// TIA Portal V17 export
// export: Created 2023-08-26T15:31:22.9849218Z, ExportSetting WithDefaults, DisplayName Totally Integrated Automation Portal, DisplayVersion V17 Update 5, DisplayName TIA Portal Openness, DisplayVersion V17 Update 5, DisplayName TIA Portal Teamcenter Gateway, DisplayVersion V17 Update 5, DisplayName TIA Portal Version Control Interface, DisplayVersion V17, DisplayName Simotion SCOUT TIA, DisplayVersion 5.4.3.0, DisplayName TIA Portal Test Suite Advanced, DisplayVersion V17 Update 1, DisplayName SIMOCODE ES, DisplayVersion V17 Update 5, DisplayName SINAMICS Startdrive Advanced, DisplayVersion V17 SP1, DisplayName SINAMICS Startdrive G130, G150, S120, S150, SINAMICS MV, S210, DisplayVersion V17 SP1, DisplayName SINAMICS Startdrive G110M, G120, G120C, G120D, G120P, G115D, DisplayVersion V17 SP1, DisplayName SIRIUS Safety ES, DisplayVersion V17 Update 5, DisplayName STEP 7 Professional, DisplayVersion V17 Update 5, DisplayName STEP 7 CFC, DisplayVersion V17 Update 1, DisplayName STEP 7 Safety, DisplayVersion V17, DisplayName WinCC Advanced, DisplayVersion V17 Update 5, DisplayName SIMATIC Visualization Architect, DisplayVersion V17 Update 5
FUNCTION "00_Only for Commissioning" : Void   // FC1, F_LAD
{ S7_Optimized_Access := 'TRUE' }
VERSION : 0.1
// Management of bypass to use during commissioning
// stored: AutoNumber true, IsIECCheckEnabled false, UDAEnableTagReadback false
BEGIN

REGION Network 1: FIRE ALARM BYPASS
   // One network per node
   // TRUE if the node is not ready to be used
   // FALSE if the node is ready
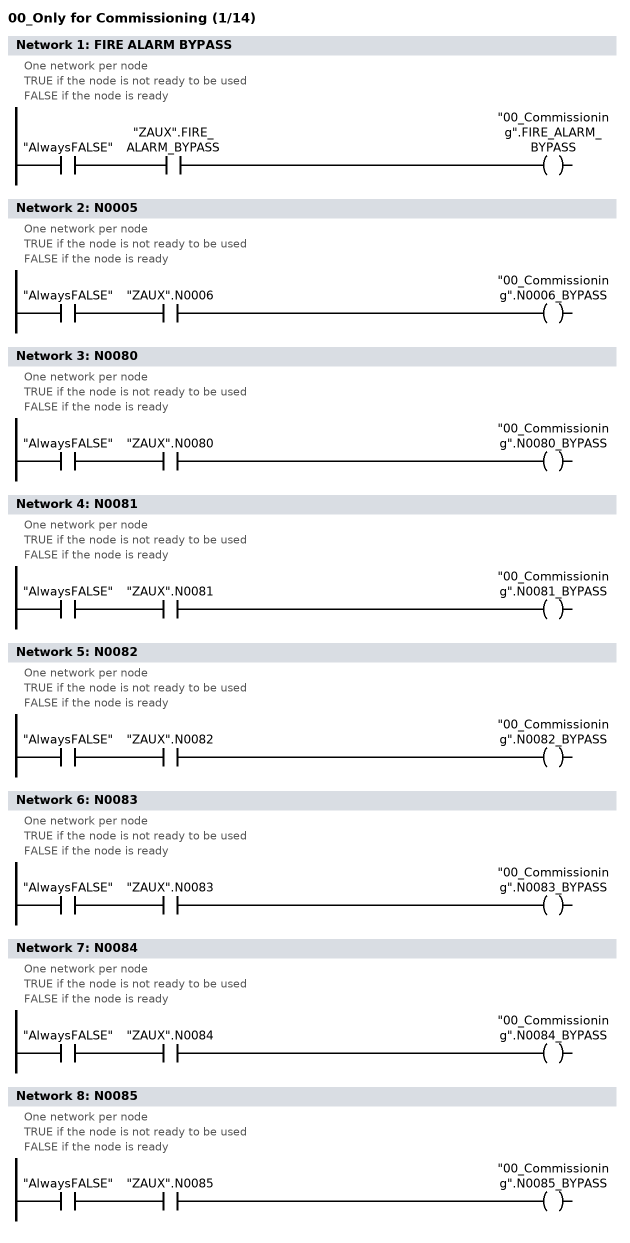
   RUNG wire#powerrail
      Contact( "AlwaysFALSE" )
      Contact( "ZAUX".FIRE_ALARM_BYPASS )
      Coil( "00_Commissioning".FIRE_ALARM_BYPASS )
   END_RUNG
   // the same network as SCL:
   "00_Commissioning".FIRE_ALARM_BYPASS := "AlwaysFALSE" AND "ZAUX".FIRE_ALARM_BYPASS;
END_REGION

REGION Network 2: N0005
   // One network per node
   // TRUE if the node is not ready to be used
   // FALSE if the node is ready
   RUNG wire#powerrail
      Contact( "AlwaysFALSE" )
      Contact( "ZAUX".N0006 )
      Coil( "00_Commissioning".N0006_BYPASS )
   END_RUNG
   // the same network as SCL:
   "00_Commissioning".N0006_BYPASS := "AlwaysFALSE" AND "ZAUX".N0006;
END_REGION

REGION Network 3: N0080
   // One network per node
   // TRUE if the node is not ready to be used
   // FALSE if the node is ready
   RUNG wire#powerrail
      Contact( "AlwaysFALSE" )
      Contact( "ZAUX".N0080 )
      Coil( "00_Commissioning".N0080_BYPASS )
   END_RUNG
   // the same network as SCL:
   "00_Commissioning".N0080_BYPASS := "AlwaysFALSE" AND "ZAUX".N0080;
END_REGION

REGION Network 4: N0081
   // One network per node
   // TRUE if the node is not ready to be used
   // FALSE if the node is ready
   RUNG wire#powerrail
      Contact( "AlwaysFALSE" )
      Contact( "ZAUX".N0081 )
      Coil( "00_Commissioning".N0081_BYPASS )
   END_RUNG
   // the same network as SCL:
   "00_Commissioning".N0081_BYPASS := "AlwaysFALSE" AND "ZAUX".N0081;
END_REGION

REGION Network 5: N0082
   // One network per node
   // TRUE if the node is not ready to be used
   // FALSE if the node is ready
   RUNG wire#powerrail
      Contact( "AlwaysFALSE" )
      Contact( "ZAUX".N0082 )
      Coil( "00_Commissioning".N0082_BYPASS )
   END_RUNG
   // the same network as SCL:
   "00_Commissioning".N0082_BYPASS := "AlwaysFALSE" AND "ZAUX".N0082;
END_REGION

REGION Network 6: N0083
   // One network per node
   // TRUE if the node is not ready to be used
   // FALSE if the node is ready
   RUNG wire#powerrail
      Contact( "AlwaysFALSE" )
      Contact( "ZAUX".N0083 )
      Coil( "00_Commissioning".N0083_BYPASS )
   END_RUNG
   // the same network as SCL:
   "00_Commissioning".N0083_BYPASS := "AlwaysFALSE" AND "ZAUX".N0083;
END_REGION

REGION Network 7: N0084
   // One network per node
   // TRUE if the node is not ready to be used
   // FALSE if the node is ready
   RUNG wire#powerrail
      Contact( "AlwaysFALSE" )
      Contact( "ZAUX".N0084 )
      Coil( "00_Commissioning".N0084_BYPASS )
   END_RUNG
   // the same network as SCL:
   "00_Commissioning".N0084_BYPASS := "AlwaysFALSE" AND "ZAUX".N0084;
END_REGION

REGION Network 8: N0085
   // One network per node
   // TRUE if the node is not ready to be used
   // FALSE if the node is ready
   RUNG wire#powerrail
      Contact( "AlwaysFALSE" )
      Contact( "ZAUX".N0085 )
      Coil( "00_Commissioning".N0085_BYPASS )
   END_RUNG
   // the same network as SCL:
   "00_Commissioning".N0085_BYPASS := "AlwaysFALSE" AND "ZAUX".N0085;
END_REGION

REGION Network 9: N0086
   // One network per node
   // TRUE if the node is not ready to be used
   // FALSE if the node is ready
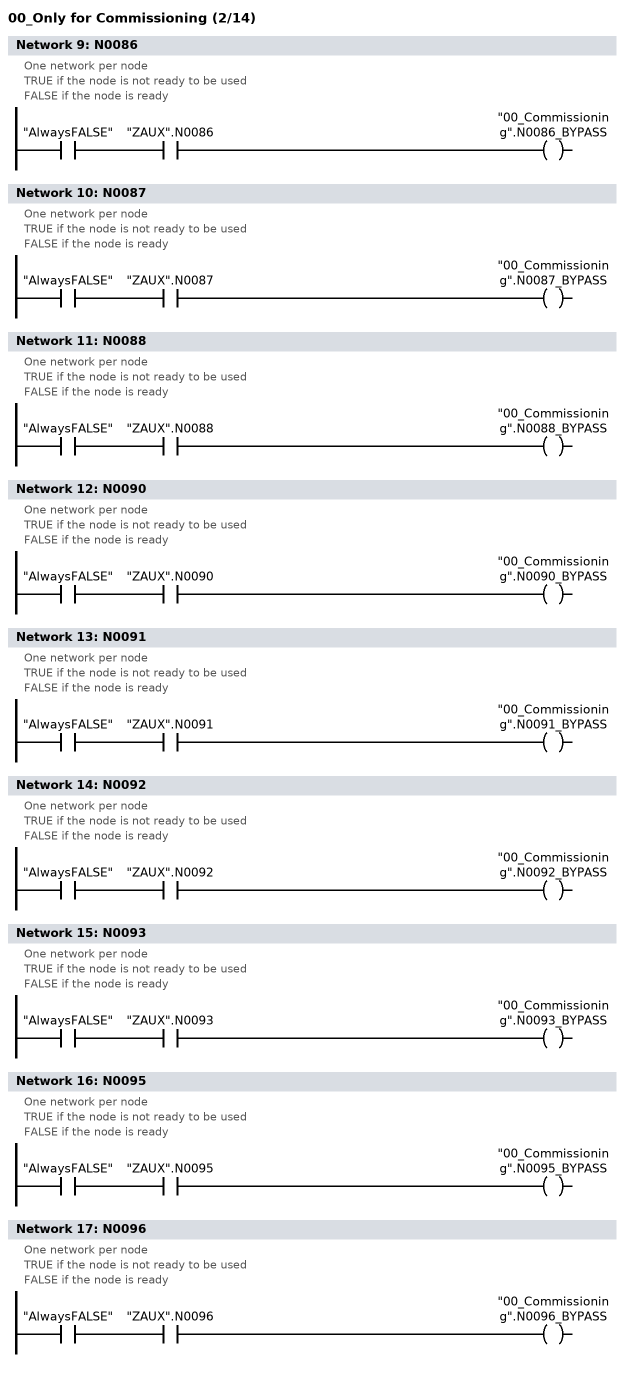
   RUNG wire#powerrail
      Contact( "AlwaysFALSE" )
      Contact( "ZAUX".N0086 )
      Coil( "00_Commissioning".N0086_BYPASS )
   END_RUNG
   // the same network as SCL:
   "00_Commissioning".N0086_BYPASS := "AlwaysFALSE" AND "ZAUX".N0086;
END_REGION

REGION Network 10: N0087
   // One network per node
   // TRUE if the node is not ready to be used
   // FALSE if the node is ready
   RUNG wire#powerrail
      Contact( "AlwaysFALSE" )
      Contact( "ZAUX".N0087 )
      Coil( "00_Commissioning".N0087_BYPASS )
   END_RUNG
   // the same network as SCL:
   "00_Commissioning".N0087_BYPASS := "AlwaysFALSE" AND "ZAUX".N0087;
END_REGION

REGION Network 11: N0088
   // One network per node
   // TRUE if the node is not ready to be used
   // FALSE if the node is ready
   RUNG wire#powerrail
      Contact( "AlwaysFALSE" )
      Contact( "ZAUX".N0088 )
      Coil( "00_Commissioning".N0088_BYPASS )
   END_RUNG
   // the same network as SCL:
   "00_Commissioning".N0088_BYPASS := "AlwaysFALSE" AND "ZAUX".N0088;
END_REGION

REGION Network 12: N0090
   // One network per node
   // TRUE if the node is not ready to be used
   // FALSE if the node is ready
   RUNG wire#powerrail
      Contact( "AlwaysFALSE" )
      Contact( "ZAUX".N0090 )
      Coil( "00_Commissioning".N0090_BYPASS )
   END_RUNG
   // the same network as SCL:
   "00_Commissioning".N0090_BYPASS := "AlwaysFALSE" AND "ZAUX".N0090;
END_REGION

REGION Network 13: N0091
   // One network per node
   // TRUE if the node is not ready to be used
   // FALSE if the node is ready
   RUNG wire#powerrail
      Contact( "AlwaysFALSE" )
      Contact( "ZAUX".N0091 )
      Coil( "00_Commissioning".N0091_BYPASS )
   END_RUNG
   // the same network as SCL:
   "00_Commissioning".N0091_BYPASS := "AlwaysFALSE" AND "ZAUX".N0091;
END_REGION

REGION Network 14: N0092
   // One network per node
   // TRUE if the node is not ready to be used
   // FALSE if the node is ready
   RUNG wire#powerrail
      Contact( "AlwaysFALSE" )
      Contact( "ZAUX".N0092 )
      Coil( "00_Commissioning".N0092_BYPASS )
   END_RUNG
   // the same network as SCL:
   "00_Commissioning".N0092_BYPASS := "AlwaysFALSE" AND "ZAUX".N0092;
END_REGION

REGION Network 15: N0093
   // One network per node
   // TRUE if the node is not ready to be used
   // FALSE if the node is ready
   RUNG wire#powerrail
      Contact( "AlwaysFALSE" )
      Contact( "ZAUX".N0093 )
      Coil( "00_Commissioning".N0093_BYPASS )
   END_RUNG
   // the same network as SCL:
   "00_Commissioning".N0093_BYPASS := "AlwaysFALSE" AND "ZAUX".N0093;
END_REGION

REGION Network 16: N0095
   // One network per node
   // TRUE if the node is not ready to be used
   // FALSE if the node is ready
   RUNG wire#powerrail
      Contact( "AlwaysFALSE" )
      Contact( "ZAUX".N0095 )
      Coil( "00_Commissioning".N0095_BYPASS )
   END_RUNG
   // the same network as SCL:
   "00_Commissioning".N0095_BYPASS := "AlwaysFALSE" AND "ZAUX".N0095;
END_REGION

REGION Network 17: N0096
   // One network per node
   // TRUE if the node is not ready to be used
   // FALSE if the node is ready
   RUNG wire#powerrail
      Contact( "AlwaysFALSE" )
      Contact( "ZAUX".N0096 )
      Coil( "00_Commissioning".N0096_BYPASS )
   END_RUNG
   // the same network as SCL:
   "00_Commissioning".N0096_BYPASS := "AlwaysFALSE" AND "ZAUX".N0096;
END_REGION

REGION Network 18: N0097
   // One network per node
   // TRUE if the node is not ready to be used
   // FALSE if the node is ready
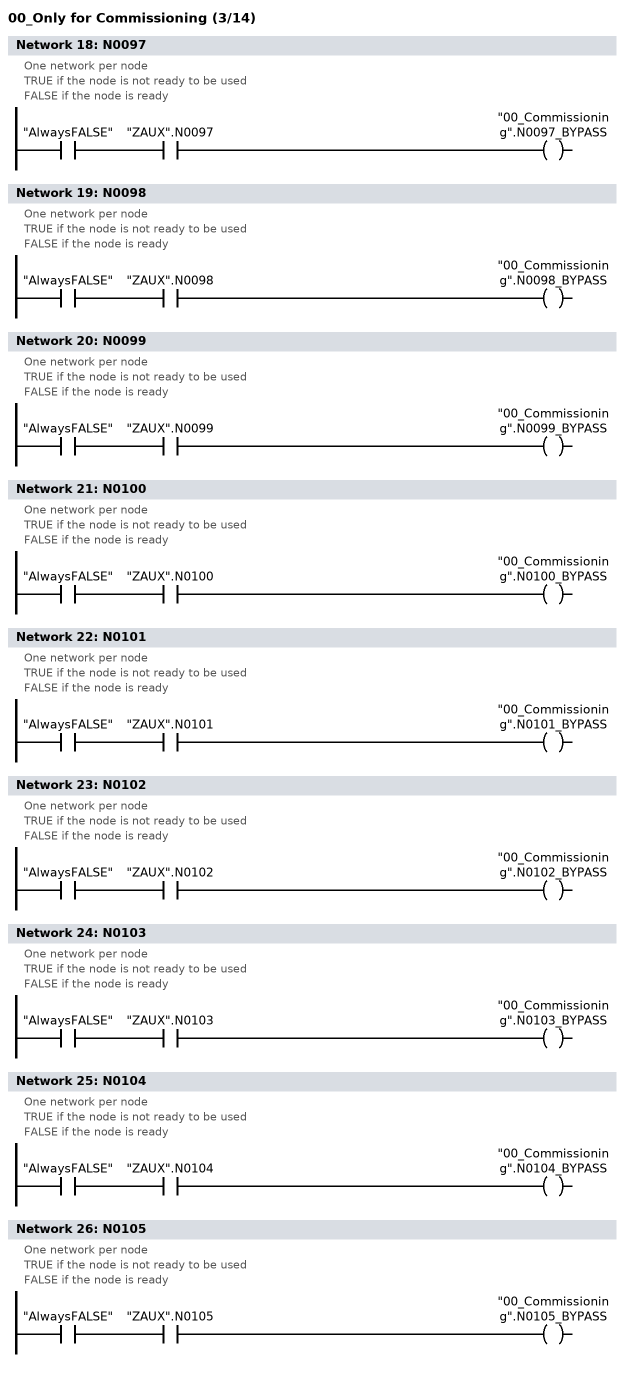
   RUNG wire#powerrail
      Contact( "AlwaysFALSE" )
      Contact( "ZAUX".N0097 )
      Coil( "00_Commissioning".N0097_BYPASS )
   END_RUNG
   // the same network as SCL:
   "00_Commissioning".N0097_BYPASS := "AlwaysFALSE" AND "ZAUX".N0097;
END_REGION

REGION Network 19: N0098
   // One network per node
   // TRUE if the node is not ready to be used
   // FALSE if the node is ready
   RUNG wire#powerrail
      Contact( "AlwaysFALSE" )
      Contact( "ZAUX".N0098 )
      Coil( "00_Commissioning".N0098_BYPASS )
   END_RUNG
   // the same network as SCL:
   "00_Commissioning".N0098_BYPASS := "AlwaysFALSE" AND "ZAUX".N0098;
END_REGION

REGION Network 20: N0099
   // One network per node
   // TRUE if the node is not ready to be used
   // FALSE if the node is ready
   RUNG wire#powerrail
      Contact( "AlwaysFALSE" )
      Contact( "ZAUX".N0099 )
      Coil( "00_Commissioning".N0099_BYPASS )
   END_RUNG
   // the same network as SCL:
   "00_Commissioning".N0099_BYPASS := "AlwaysFALSE" AND "ZAUX".N0099;
END_REGION

REGION Network 21: N0100
   // One network per node
   // TRUE if the node is not ready to be used
   // FALSE if the node is ready
   RUNG wire#powerrail
      Contact( "AlwaysFALSE" )
      Contact( "ZAUX".N0100 )
      Coil( "00_Commissioning".N0100_BYPASS )
   END_RUNG
   // the same network as SCL:
   "00_Commissioning".N0100_BYPASS := "AlwaysFALSE" AND "ZAUX".N0100;
END_REGION

REGION Network 22: N0101
   // One network per node
   // TRUE if the node is not ready to be used
   // FALSE if the node is ready
   RUNG wire#powerrail
      Contact( "AlwaysFALSE" )
      Contact( "ZAUX".N0101 )
      Coil( "00_Commissioning".N0101_BYPASS )
   END_RUNG
   // the same network as SCL:
   "00_Commissioning".N0101_BYPASS := "AlwaysFALSE" AND "ZAUX".N0101;
END_REGION

REGION Network 23: N0102
   // One network per node
   // TRUE if the node is not ready to be used
   // FALSE if the node is ready
   RUNG wire#powerrail
      Contact( "AlwaysFALSE" )
      Contact( "ZAUX".N0102 )
      Coil( "00_Commissioning".N0102_BYPASS )
   END_RUNG
   // the same network as SCL:
   "00_Commissioning".N0102_BYPASS := "AlwaysFALSE" AND "ZAUX".N0102;
END_REGION

REGION Network 24: N0103
   // One network per node
   // TRUE if the node is not ready to be used
   // FALSE if the node is ready
   RUNG wire#powerrail
      Contact( "AlwaysFALSE" )
      Contact( "ZAUX".N0103 )
      Coil( "00_Commissioning".N0103_BYPASS )
   END_RUNG
   // the same network as SCL:
   "00_Commissioning".N0103_BYPASS := "AlwaysFALSE" AND "ZAUX".N0103;
END_REGION

REGION Network 25: N0104
   // One network per node
   // TRUE if the node is not ready to be used
   // FALSE if the node is ready
   RUNG wire#powerrail
      Contact( "AlwaysFALSE" )
      Contact( "ZAUX".N0104 )
      Coil( "00_Commissioning".N0104_BYPASS )
   END_RUNG
   // the same network as SCL:
   "00_Commissioning".N0104_BYPASS := "AlwaysFALSE" AND "ZAUX".N0104;
END_REGION

REGION Network 26: N0105
   // One network per node
   // TRUE if the node is not ready to be used
   // FALSE if the node is ready
   RUNG wire#powerrail
      Contact( "AlwaysFALSE" )
      Contact( "ZAUX".N0105 )
      Coil( "00_Commissioning".N0105_BYPASS )
   END_RUNG
   // the same network as SCL:
   "00_Commissioning".N0105_BYPASS := "AlwaysFALSE" AND "ZAUX".N0105;
END_REGION

REGION Network 27: N0106
   // One network per node
   // TRUE if the node is not ready to be used
   // FALSE if the node is ready
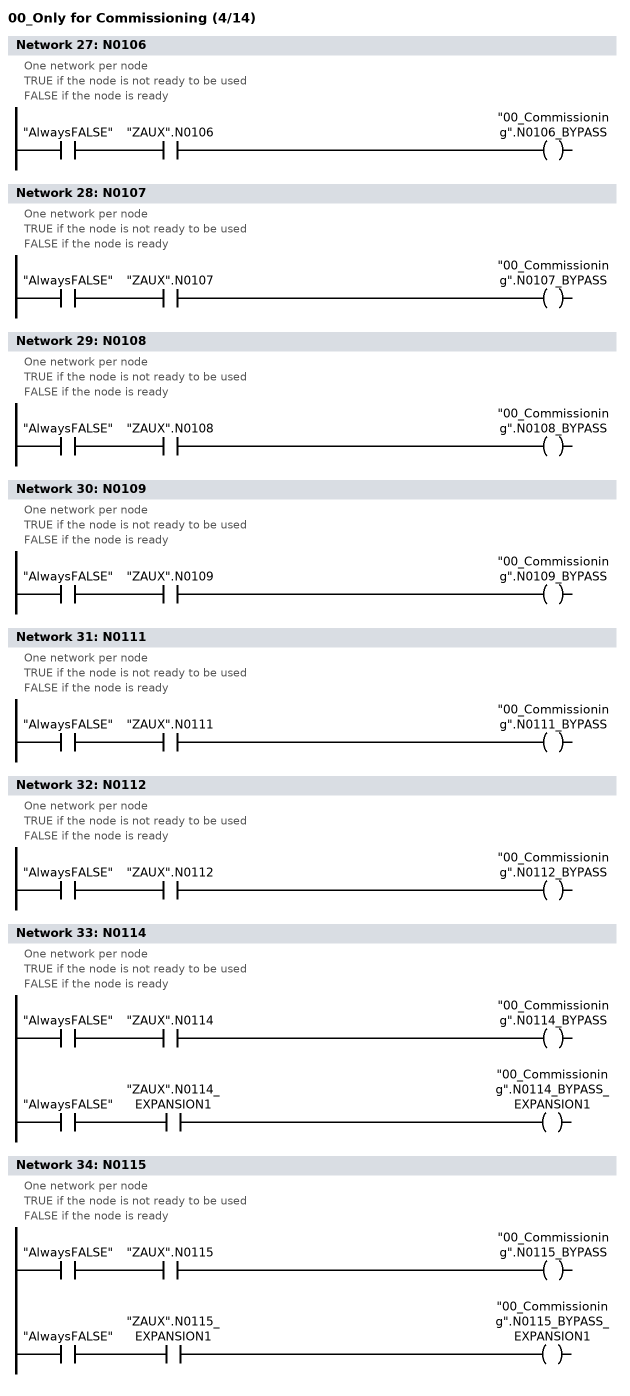
   RUNG wire#powerrail
      Contact( "AlwaysFALSE" )
      Contact( "ZAUX".N0106 )
      Coil( "00_Commissioning".N0106_BYPASS )
   END_RUNG
   // the same network as SCL:
   "00_Commissioning".N0106_BYPASS := "AlwaysFALSE" AND "ZAUX".N0106;
END_REGION

REGION Network 28: N0107
   // One network per node
   // TRUE if the node is not ready to be used
   // FALSE if the node is ready
   RUNG wire#powerrail
      Contact( "AlwaysFALSE" )
      Contact( "ZAUX".N0107 )
      Coil( "00_Commissioning".N0107_BYPASS )
   END_RUNG
   // the same network as SCL:
   "00_Commissioning".N0107_BYPASS := "AlwaysFALSE" AND "ZAUX".N0107;
END_REGION

REGION Network 29: N0108
   // One network per node
   // TRUE if the node is not ready to be used
   // FALSE if the node is ready
   RUNG wire#powerrail
      Contact( "AlwaysFALSE" )
      Contact( "ZAUX".N0108 )
      Coil( "00_Commissioning".N0108_BYPASS )
   END_RUNG
   // the same network as SCL:
   "00_Commissioning".N0108_BYPASS := "AlwaysFALSE" AND "ZAUX".N0108;
END_REGION

REGION Network 30: N0109
   // One network per node
   // TRUE if the node is not ready to be used
   // FALSE if the node is ready
   RUNG wire#powerrail
      Contact( "AlwaysFALSE" )
      Contact( "ZAUX".N0109 )
      Coil( "00_Commissioning".N0109_BYPASS )
   END_RUNG
   // the same network as SCL:
   "00_Commissioning".N0109_BYPASS := "AlwaysFALSE" AND "ZAUX".N0109;
END_REGION

REGION Network 31: N0111
   // One network per node
   // TRUE if the node is not ready to be used
   // FALSE if the node is ready
   RUNG wire#powerrail
      Contact( "AlwaysFALSE" )
      Contact( "ZAUX".N0111 )
      Coil( "00_Commissioning".N0111_BYPASS )
   END_RUNG
   // the same network as SCL:
   "00_Commissioning".N0111_BYPASS := "AlwaysFALSE" AND "ZAUX".N0111;
END_REGION

REGION Network 32: N0112
   // One network per node
   // TRUE if the node is not ready to be used
   // FALSE if the node is ready
   RUNG wire#powerrail
      Contact( "AlwaysFALSE" )
      Contact( "ZAUX".N0112 )
      Coil( "00_Commissioning".N0112_BYPASS )
   END_RUNG
   // the same network as SCL:
   "00_Commissioning".N0112_BYPASS := "AlwaysFALSE" AND "ZAUX".N0112;
END_REGION

REGION Network 33: N0114
   // One network per node
   // TRUE if the node is not ready to be used
   // FALSE if the node is ready
   RUNG wire#powerrail
      Contact( "AlwaysFALSE" )
      Contact( "ZAUX".N0114 )
      Coil( "00_Commissioning".N0114_BYPASS )
   END_RUNG
   RUNG wire#powerrail
      Contact( "AlwaysFALSE" )
      Contact( "ZAUX".N0114_EXPANSION1 )
      Coil( "00_Commissioning".N0114_BYPASS_EXPANSION1 )
   END_RUNG
   // the same network as SCL:
   "00_Commissioning".N0114_BYPASS := "AlwaysFALSE" AND "ZAUX".N0114;
   "00_Commissioning".N0114_BYPASS_EXPANSION1 := "AlwaysFALSE" AND "ZAUX".N0114_EXPANSION1;
END_REGION

REGION Network 34: N0115
   // One network per node
   // TRUE if the node is not ready to be used
   // FALSE if the node is ready
   RUNG wire#powerrail
      Contact( "AlwaysFALSE" )
      Contact( "ZAUX".N0115 )
      Coil( "00_Commissioning".N0115_BYPASS )
   END_RUNG
   RUNG wire#powerrail
      Contact( "AlwaysFALSE" )
      Contact( "ZAUX".N0115_EXPANSION1 )
      Coil( "00_Commissioning".N0115_BYPASS_EXPANSION1 )
   END_RUNG
   // the same network as SCL:
   "00_Commissioning".N0115_BYPASS := "AlwaysFALSE" AND "ZAUX".N0115;
   "00_Commissioning".N0115_BYPASS_EXPANSION1 := "AlwaysFALSE" AND "ZAUX".N0115_EXPANSION1;
END_REGION

REGION Network 35: N0116
   // One network per node
   // TRUE if the node is not ready to be used
   // FALSE if the node is ready
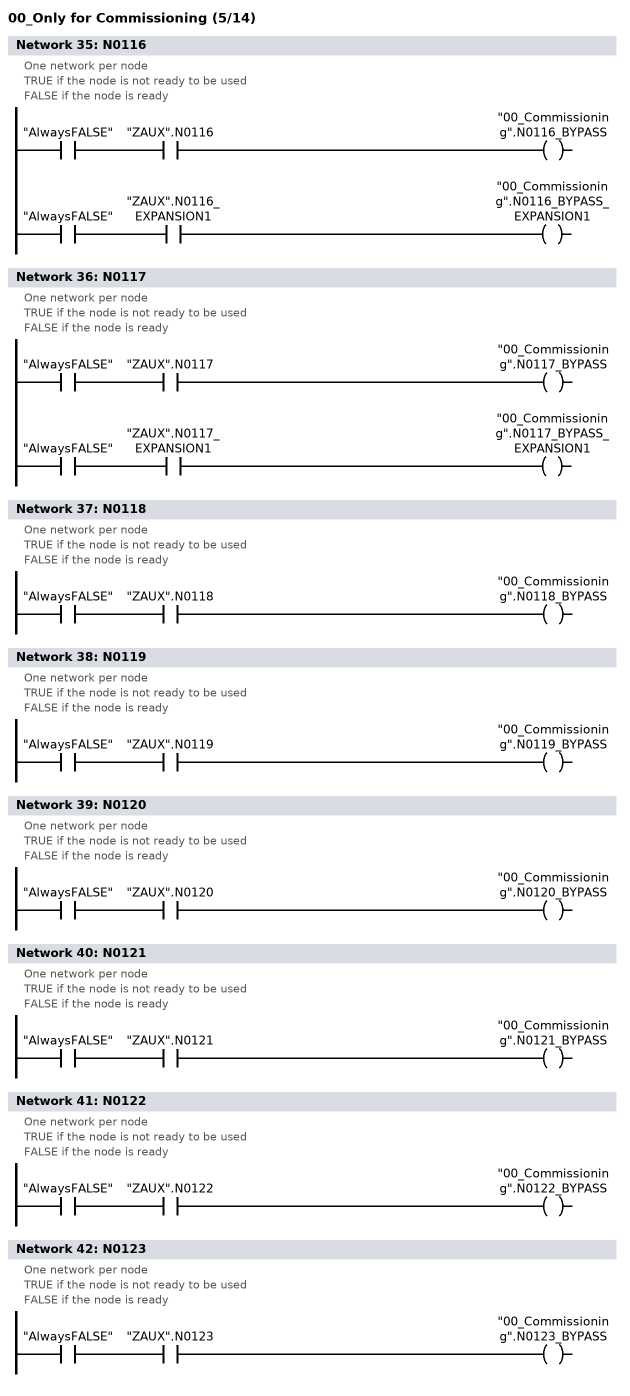
   RUNG wire#powerrail
      Contact( "AlwaysFALSE" )
      Contact( "ZAUX".N0116 )
      Coil( "00_Commissioning".N0116_BYPASS )
   END_RUNG
   RUNG wire#powerrail
      Contact( "AlwaysFALSE" )
      Contact( "ZAUX".N0116_EXPANSION1 )
      Coil( "00_Commissioning".N0116_BYPASS_EXPANSION1 )
   END_RUNG
   // the same network as SCL:
   "00_Commissioning".N0116_BYPASS := "AlwaysFALSE" AND "ZAUX".N0116;
   "00_Commissioning".N0116_BYPASS_EXPANSION1 := "AlwaysFALSE" AND "ZAUX".N0116_EXPANSION1;
END_REGION

REGION Network 36: N0117
   // One network per node
   // TRUE if the node is not ready to be used
   // FALSE if the node is ready
   RUNG wire#powerrail
      Contact( "AlwaysFALSE" )
      Contact( "ZAUX".N0117 )
      Coil( "00_Commissioning".N0117_BYPASS )
   END_RUNG
   RUNG wire#powerrail
      Contact( "AlwaysFALSE" )
      Contact( "ZAUX".N0117_EXPANSION1 )
      Coil( "00_Commissioning".N0117_BYPASS_EXPANSION1 )
   END_RUNG
   // the same network as SCL:
   "00_Commissioning".N0117_BYPASS := "AlwaysFALSE" AND "ZAUX".N0117;
   "00_Commissioning".N0117_BYPASS_EXPANSION1 := "AlwaysFALSE" AND "ZAUX".N0117_EXPANSION1;
END_REGION

REGION Network 37: N0118
   // One network per node
   // TRUE if the node is not ready to be used
   // FALSE if the node is ready
   RUNG wire#powerrail
      Contact( "AlwaysFALSE" )
      Contact( "ZAUX".N0118 )
      Coil( "00_Commissioning".N0118_BYPASS )
   END_RUNG
   // the same network as SCL:
   "00_Commissioning".N0118_BYPASS := "AlwaysFALSE" AND "ZAUX".N0118;
END_REGION

REGION Network 38: N0119
   // One network per node
   // TRUE if the node is not ready to be used
   // FALSE if the node is ready
   RUNG wire#powerrail
      Contact( "AlwaysFALSE" )
      Contact( "ZAUX".N0119 )
      Coil( "00_Commissioning".N0119_BYPASS )
   END_RUNG
   // the same network as SCL:
   "00_Commissioning".N0119_BYPASS := "AlwaysFALSE" AND "ZAUX".N0119;
END_REGION

REGION Network 39: N0120
   // One network per node
   // TRUE if the node is not ready to be used
   // FALSE if the node is ready
   RUNG wire#powerrail
      Contact( "AlwaysFALSE" )
      Contact( "ZAUX".N0120 )
      Coil( "00_Commissioning".N0120_BYPASS )
   END_RUNG
   // the same network as SCL:
   "00_Commissioning".N0120_BYPASS := "AlwaysFALSE" AND "ZAUX".N0120;
END_REGION

REGION Network 40: N0121
   // One network per node
   // TRUE if the node is not ready to be used
   // FALSE if the node is ready
   RUNG wire#powerrail
      Contact( "AlwaysFALSE" )
      Contact( "ZAUX".N0121 )
      Coil( "00_Commissioning".N0121_BYPASS )
   END_RUNG
   // the same network as SCL:
   "00_Commissioning".N0121_BYPASS := "AlwaysFALSE" AND "ZAUX".N0121;
END_REGION

REGION Network 41: N0122
   // One network per node
   // TRUE if the node is not ready to be used
   // FALSE if the node is ready
   RUNG wire#powerrail
      Contact( "AlwaysFALSE" )
      Contact( "ZAUX".N0122 )
      Coil( "00_Commissioning".N0122_BYPASS )
   END_RUNG
   // the same network as SCL:
   "00_Commissioning".N0122_BYPASS := "AlwaysFALSE" AND "ZAUX".N0122;
END_REGION

REGION Network 42: N0123
   // One network per node
   // TRUE if the node is not ready to be used
   // FALSE if the node is ready
   RUNG wire#powerrail
      Contact( "AlwaysFALSE" )
      Contact( "ZAUX".N0123 )
      Coil( "00_Commissioning".N0123_BYPASS )
   END_RUNG
   // the same network as SCL:
   "00_Commissioning".N0123_BYPASS := "AlwaysFALSE" AND "ZAUX".N0123;
END_REGION

REGION Network 43: N0124
   // One network per node
   // TRUE if the node is not ready to be used
   // FALSE if the node is ready
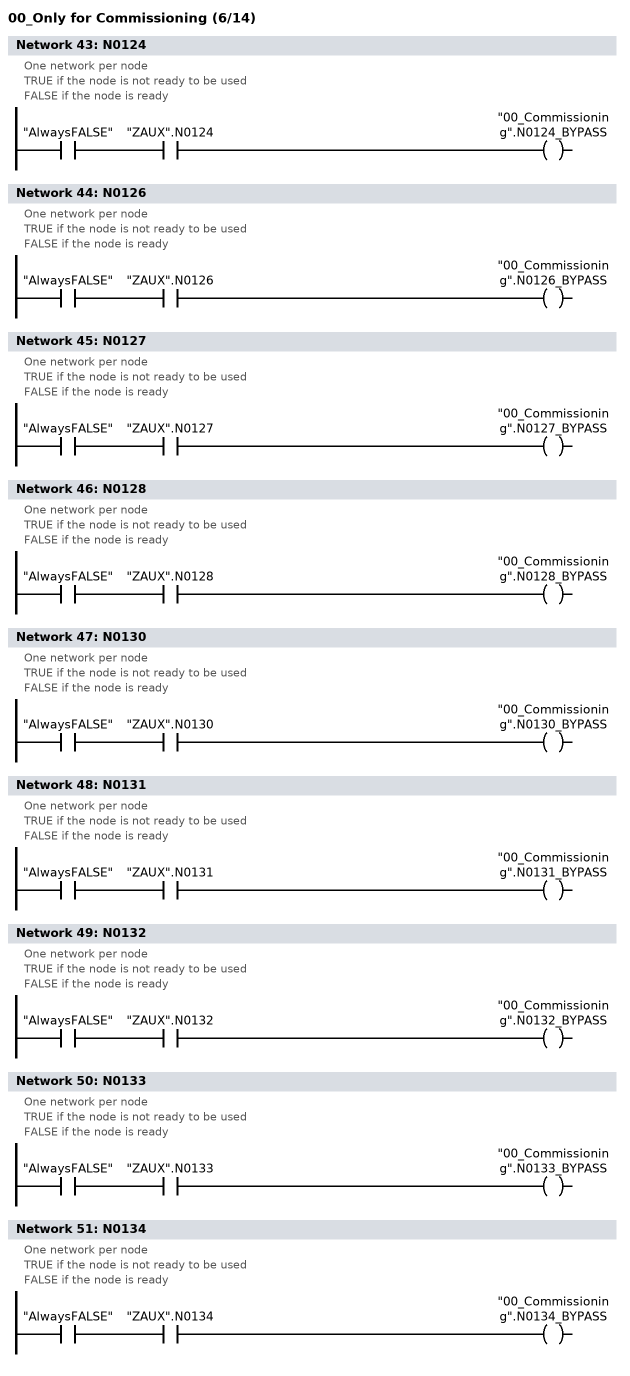
   RUNG wire#powerrail
      Contact( "AlwaysFALSE" )
      Contact( "ZAUX".N0124 )
      Coil( "00_Commissioning".N0124_BYPASS )
   END_RUNG
   // the same network as SCL:
   "00_Commissioning".N0124_BYPASS := "AlwaysFALSE" AND "ZAUX".N0124;
END_REGION

REGION Network 44: N0126
   // One network per node
   // TRUE if the node is not ready to be used
   // FALSE if the node is ready
   RUNG wire#powerrail
      Contact( "AlwaysFALSE" )
      Contact( "ZAUX".N0126 )
      Coil( "00_Commissioning".N0126_BYPASS )
   END_RUNG
   // the same network as SCL:
   "00_Commissioning".N0126_BYPASS := "AlwaysFALSE" AND "ZAUX".N0126;
END_REGION

REGION Network 45: N0127
   // One network per node
   // TRUE if the node is not ready to be used
   // FALSE if the node is ready
   RUNG wire#powerrail
      Contact( "AlwaysFALSE" )
      Contact( "ZAUX".N0127 )
      Coil( "00_Commissioning".N0127_BYPASS )
   END_RUNG
   // the same network as SCL:
   "00_Commissioning".N0127_BYPASS := "AlwaysFALSE" AND "ZAUX".N0127;
END_REGION

REGION Network 46: N0128
   // One network per node
   // TRUE if the node is not ready to be used
   // FALSE if the node is ready
   RUNG wire#powerrail
      Contact( "AlwaysFALSE" )
      Contact( "ZAUX".N0128 )
      Coil( "00_Commissioning".N0128_BYPASS )
   END_RUNG
   // the same network as SCL:
   "00_Commissioning".N0128_BYPASS := "AlwaysFALSE" AND "ZAUX".N0128;
END_REGION

REGION Network 47: N0130
   // One network per node
   // TRUE if the node is not ready to be used
   // FALSE if the node is ready
   RUNG wire#powerrail
      Contact( "AlwaysFALSE" )
      Contact( "ZAUX".N0130 )
      Coil( "00_Commissioning".N0130_BYPASS )
   END_RUNG
   // the same network as SCL:
   "00_Commissioning".N0130_BYPASS := "AlwaysFALSE" AND "ZAUX".N0130;
END_REGION

REGION Network 48: N0131
   // One network per node
   // TRUE if the node is not ready to be used
   // FALSE if the node is ready
   RUNG wire#powerrail
      Contact( "AlwaysFALSE" )
      Contact( "ZAUX".N0131 )
      Coil( "00_Commissioning".N0131_BYPASS )
   END_RUNG
   // the same network as SCL:
   "00_Commissioning".N0131_BYPASS := "AlwaysFALSE" AND "ZAUX".N0131;
END_REGION

REGION Network 49: N0132
   // One network per node
   // TRUE if the node is not ready to be used
   // FALSE if the node is ready
   RUNG wire#powerrail
      Contact( "AlwaysFALSE" )
      Contact( "ZAUX".N0132 )
      Coil( "00_Commissioning".N0132_BYPASS )
   END_RUNG
   // the same network as SCL:
   "00_Commissioning".N0132_BYPASS := "AlwaysFALSE" AND "ZAUX".N0132;
END_REGION

REGION Network 50: N0133
   // One network per node
   // TRUE if the node is not ready to be used
   // FALSE if the node is ready
   RUNG wire#powerrail
      Contact( "AlwaysFALSE" )
      Contact( "ZAUX".N0133 )
      Coil( "00_Commissioning".N0133_BYPASS )
   END_RUNG
   // the same network as SCL:
   "00_Commissioning".N0133_BYPASS := "AlwaysFALSE" AND "ZAUX".N0133;
END_REGION

REGION Network 51: N0134
   // One network per node
   // TRUE if the node is not ready to be used
   // FALSE if the node is ready
   RUNG wire#powerrail
      Contact( "AlwaysFALSE" )
      Contact( "ZAUX".N0134 )
      Coil( "00_Commissioning".N0134_BYPASS )
   END_RUNG
   // the same network as SCL:
   "00_Commissioning".N0134_BYPASS := "AlwaysFALSE" AND "ZAUX".N0134;
END_REGION

REGION Network 52: N0137
   // One network per node
   // TRUE if the node is not ready to be used
   // FALSE if the node is ready
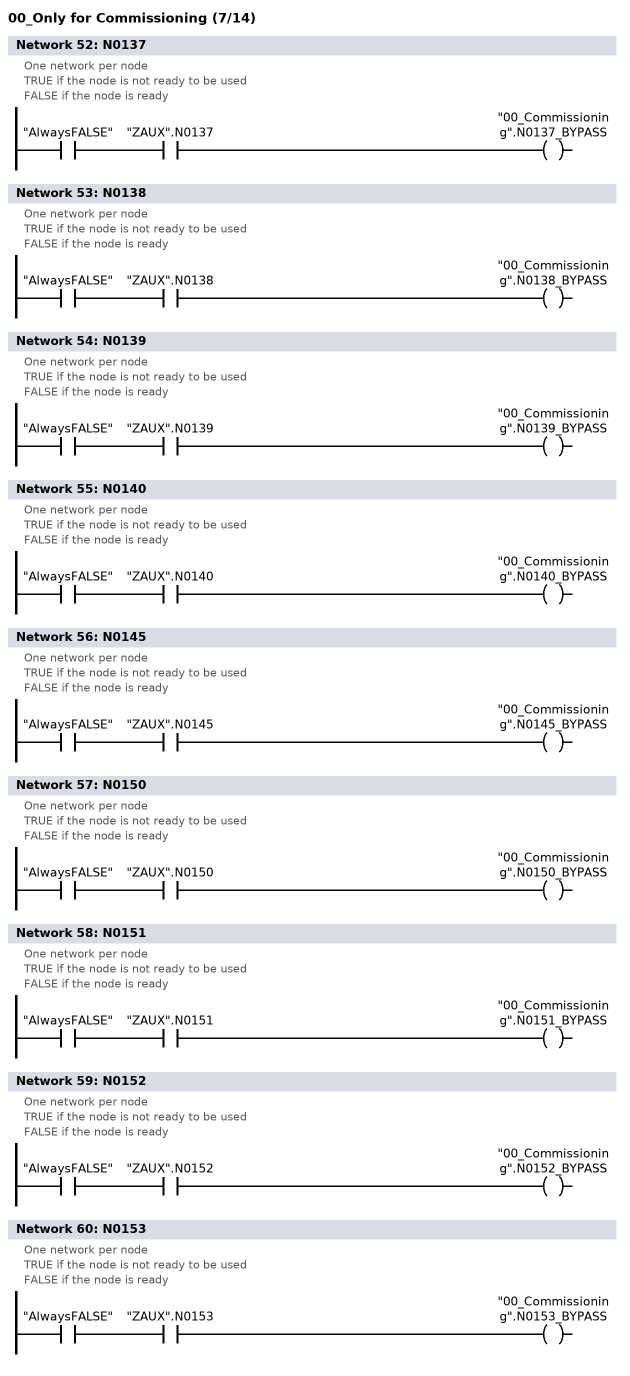
   RUNG wire#powerrail
      Contact( "AlwaysFALSE" )
      Contact( "ZAUX".N0137 )
      Coil( "00_Commissioning".N0137_BYPASS )
   END_RUNG
   // the same network as SCL:
   "00_Commissioning".N0137_BYPASS := "AlwaysFALSE" AND "ZAUX".N0137;
END_REGION

REGION Network 53: N0138
   // One network per node
   // TRUE if the node is not ready to be used
   // FALSE if the node is ready
   RUNG wire#powerrail
      Contact( "AlwaysFALSE" )
      Contact( "ZAUX".N0138 )
      Coil( "00_Commissioning".N0138_BYPASS )
   END_RUNG
   // the same network as SCL:
   "00_Commissioning".N0138_BYPASS := "AlwaysFALSE" AND "ZAUX".N0138;
END_REGION

REGION Network 54: N0139
   // One network per node
   // TRUE if the node is not ready to be used
   // FALSE if the node is ready
   RUNG wire#powerrail
      Contact( "AlwaysFALSE" )
      Contact( "ZAUX".N0139 )
      Coil( "00_Commissioning".N0139_BYPASS )
   END_RUNG
   // the same network as SCL:
   "00_Commissioning".N0139_BYPASS := "AlwaysFALSE" AND "ZAUX".N0139;
END_REGION

REGION Network 55: N0140
   // One network per node
   // TRUE if the node is not ready to be used
   // FALSE if the node is ready
   RUNG wire#powerrail
      Contact( "AlwaysFALSE" )
      Contact( "ZAUX".N0140 )
      Coil( "00_Commissioning".N0140_BYPASS )
   END_RUNG
   // the same network as SCL:
   "00_Commissioning".N0140_BYPASS := "AlwaysFALSE" AND "ZAUX".N0140;
END_REGION

REGION Network 56: N0145
   // One network per node
   // TRUE if the node is not ready to be used
   // FALSE if the node is ready
   RUNG wire#powerrail
      Contact( "AlwaysFALSE" )
      Contact( "ZAUX".N0145 )
      Coil( "00_Commissioning".N0145_BYPASS )
   END_RUNG
   // the same network as SCL:
   "00_Commissioning".N0145_BYPASS := "AlwaysFALSE" AND "ZAUX".N0145;
END_REGION

REGION Network 57: N0150
   // One network per node
   // TRUE if the node is not ready to be used
   // FALSE if the node is ready
   RUNG wire#powerrail
      Contact( "AlwaysFALSE" )
      Contact( "ZAUX".N0150 )
      Coil( "00_Commissioning".N0150_BYPASS )
   END_RUNG
   // the same network as SCL:
   "00_Commissioning".N0150_BYPASS := "AlwaysFALSE" AND "ZAUX".N0150;
END_REGION

REGION Network 58: N0151
   // One network per node
   // TRUE if the node is not ready to be used
   // FALSE if the node is ready
   RUNG wire#powerrail
      Contact( "AlwaysFALSE" )
      Contact( "ZAUX".N0151 )
      Coil( "00_Commissioning".N0151_BYPASS )
   END_RUNG
   // the same network as SCL:
   "00_Commissioning".N0151_BYPASS := "AlwaysFALSE" AND "ZAUX".N0151;
END_REGION

REGION Network 59: N0152
   // One network per node
   // TRUE if the node is not ready to be used
   // FALSE if the node is ready
   RUNG wire#powerrail
      Contact( "AlwaysFALSE" )
      Contact( "ZAUX".N0152 )
      Coil( "00_Commissioning".N0152_BYPASS )
   END_RUNG
   // the same network as SCL:
   "00_Commissioning".N0152_BYPASS := "AlwaysFALSE" AND "ZAUX".N0152;
END_REGION

REGION Network 60: N0153
   // One network per node
   // TRUE if the node is not ready to be used
   // FALSE if the node is ready
   RUNG wire#powerrail
      Contact( "AlwaysFALSE" )
      Contact( "ZAUX".N0153 )
      Coil( "00_Commissioning".N0153_BYPASS )
   END_RUNG
   // the same network as SCL:
   "00_Commissioning".N0153_BYPASS := "AlwaysFALSE" AND "ZAUX".N0153;
END_REGION

REGION Network 61: N0154
   // One network per node
   // TRUE if the node is not ready to be used
   // FALSE if the node is ready
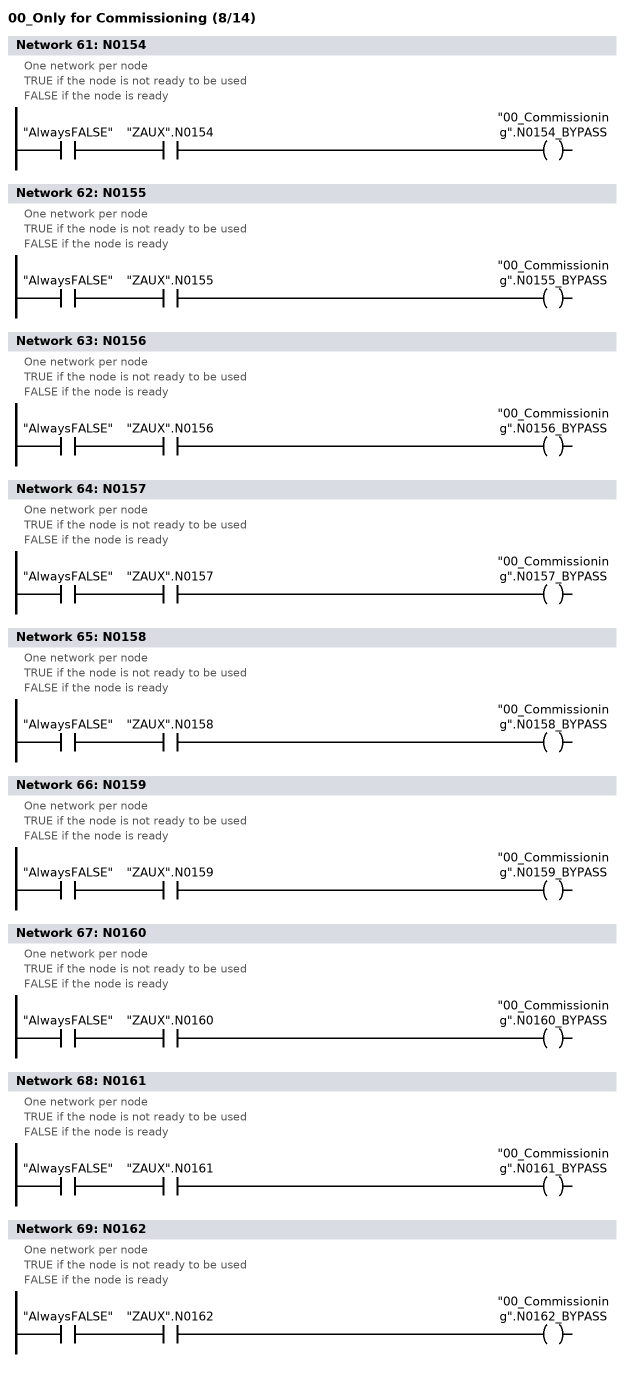
   RUNG wire#powerrail
      Contact( "AlwaysFALSE" )
      Contact( "ZAUX".N0154 )
      Coil( "00_Commissioning".N0154_BYPASS )
   END_RUNG
   // the same network as SCL:
   "00_Commissioning".N0154_BYPASS := "AlwaysFALSE" AND "ZAUX".N0154;
END_REGION

REGION Network 62: N0155
   // One network per node
   // TRUE if the node is not ready to be used
   // FALSE if the node is ready
   RUNG wire#powerrail
      Contact( "AlwaysFALSE" )
      Contact( "ZAUX".N0155 )
      Coil( "00_Commissioning".N0155_BYPASS )
   END_RUNG
   // the same network as SCL:
   "00_Commissioning".N0155_BYPASS := "AlwaysFALSE" AND "ZAUX".N0155;
END_REGION

REGION Network 63: N0156
   // One network per node
   // TRUE if the node is not ready to be used
   // FALSE if the node is ready
   RUNG wire#powerrail
      Contact( "AlwaysFALSE" )
      Contact( "ZAUX".N0156 )
      Coil( "00_Commissioning".N0156_BYPASS )
   END_RUNG
   // the same network as SCL:
   "00_Commissioning".N0156_BYPASS := "AlwaysFALSE" AND "ZAUX".N0156;
END_REGION

REGION Network 64: N0157
   // One network per node
   // TRUE if the node is not ready to be used
   // FALSE if the node is ready
   RUNG wire#powerrail
      Contact( "AlwaysFALSE" )
      Contact( "ZAUX".N0157 )
      Coil( "00_Commissioning".N0157_BYPASS )
   END_RUNG
   // the same network as SCL:
   "00_Commissioning".N0157_BYPASS := "AlwaysFALSE" AND "ZAUX".N0157;
END_REGION

REGION Network 65: N0158
   // One network per node
   // TRUE if the node is not ready to be used
   // FALSE if the node is ready
   RUNG wire#powerrail
      Contact( "AlwaysFALSE" )
      Contact( "ZAUX".N0158 )
      Coil( "00_Commissioning".N0158_BYPASS )
   END_RUNG
   // the same network as SCL:
   "00_Commissioning".N0158_BYPASS := "AlwaysFALSE" AND "ZAUX".N0158;
END_REGION

REGION Network 66: N0159
   // One network per node
   // TRUE if the node is not ready to be used
   // FALSE if the node is ready
   RUNG wire#powerrail
      Contact( "AlwaysFALSE" )
      Contact( "ZAUX".N0159 )
      Coil( "00_Commissioning".N0159_BYPASS )
   END_RUNG
   // the same network as SCL:
   "00_Commissioning".N0159_BYPASS := "AlwaysFALSE" AND "ZAUX".N0159;
END_REGION

REGION Network 67: N0160
   // One network per node
   // TRUE if the node is not ready to be used
   // FALSE if the node is ready
   RUNG wire#powerrail
      Contact( "AlwaysFALSE" )
      Contact( "ZAUX".N0160 )
      Coil( "00_Commissioning".N0160_BYPASS )
   END_RUNG
   // the same network as SCL:
   "00_Commissioning".N0160_BYPASS := "AlwaysFALSE" AND "ZAUX".N0160;
END_REGION

REGION Network 68: N0161
   // One network per node
   // TRUE if the node is not ready to be used
   // FALSE if the node is ready
   RUNG wire#powerrail
      Contact( "AlwaysFALSE" )
      Contact( "ZAUX".N0161 )
      Coil( "00_Commissioning".N0161_BYPASS )
   END_RUNG
   // the same network as SCL:
   "00_Commissioning".N0161_BYPASS := "AlwaysFALSE" AND "ZAUX".N0161;
END_REGION

REGION Network 69: N0162
   // One network per node
   // TRUE if the node is not ready to be used
   // FALSE if the node is ready
   RUNG wire#powerrail
      Contact( "AlwaysFALSE" )
      Contact( "ZAUX".N0162 )
      Coil( "00_Commissioning".N0162_BYPASS )
   END_RUNG
   // the same network as SCL:
   "00_Commissioning".N0162_BYPASS := "AlwaysFALSE" AND "ZAUX".N0162;
END_REGION

REGION Network 70: N0163
   // One network per node
   // TRUE if the node is not ready to be used
   // FALSE if the node is ready
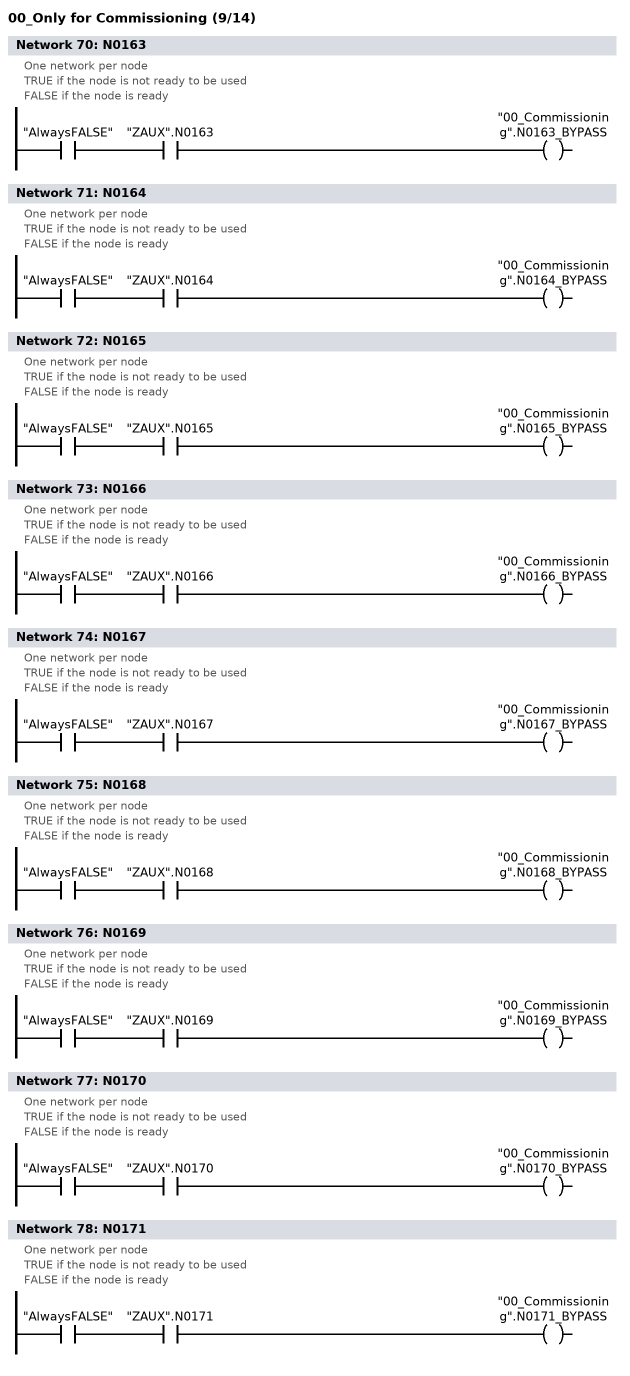
   RUNG wire#powerrail
      Contact( "AlwaysFALSE" )
      Contact( "ZAUX".N0163 )
      Coil( "00_Commissioning".N0163_BYPASS )
   END_RUNG
   // the same network as SCL:
   "00_Commissioning".N0163_BYPASS := "AlwaysFALSE" AND "ZAUX".N0163;
END_REGION

REGION Network 71: N0164
   // One network per node
   // TRUE if the node is not ready to be used
   // FALSE if the node is ready
   RUNG wire#powerrail
      Contact( "AlwaysFALSE" )
      Contact( "ZAUX".N0164 )
      Coil( "00_Commissioning".N0164_BYPASS )
   END_RUNG
   // the same network as SCL:
   "00_Commissioning".N0164_BYPASS := "AlwaysFALSE" AND "ZAUX".N0164;
END_REGION

REGION Network 72: N0165
   // One network per node
   // TRUE if the node is not ready to be used
   // FALSE if the node is ready
   RUNG wire#powerrail
      Contact( "AlwaysFALSE" )
      Contact( "ZAUX".N0165 )
      Coil( "00_Commissioning".N0165_BYPASS )
   END_RUNG
   // the same network as SCL:
   "00_Commissioning".N0165_BYPASS := "AlwaysFALSE" AND "ZAUX".N0165;
END_REGION

REGION Network 73: N0166
   // One network per node
   // TRUE if the node is not ready to be used
   // FALSE if the node is ready
   RUNG wire#powerrail
      Contact( "AlwaysFALSE" )
      Contact( "ZAUX".N0166 )
      Coil( "00_Commissioning".N0166_BYPASS )
   END_RUNG
   // the same network as SCL:
   "00_Commissioning".N0166_BYPASS := "AlwaysFALSE" AND "ZAUX".N0166;
END_REGION

REGION Network 74: N0167
   // One network per node
   // TRUE if the node is not ready to be used
   // FALSE if the node is ready
   RUNG wire#powerrail
      Contact( "AlwaysFALSE" )
      Contact( "ZAUX".N0167 )
      Coil( "00_Commissioning".N0167_BYPASS )
   END_RUNG
   // the same network as SCL:
   "00_Commissioning".N0167_BYPASS := "AlwaysFALSE" AND "ZAUX".N0167;
END_REGION

REGION Network 75: N0168
   // One network per node
   // TRUE if the node is not ready to be used
   // FALSE if the node is ready
   RUNG wire#powerrail
      Contact( "AlwaysFALSE" )
      Contact( "ZAUX".N0168 )
      Coil( "00_Commissioning".N0168_BYPASS )
   END_RUNG
   // the same network as SCL:
   "00_Commissioning".N0168_BYPASS := "AlwaysFALSE" AND "ZAUX".N0168;
END_REGION

REGION Network 76: N0169
   // One network per node
   // TRUE if the node is not ready to be used
   // FALSE if the node is ready
   RUNG wire#powerrail
      Contact( "AlwaysFALSE" )
      Contact( "ZAUX".N0169 )
      Coil( "00_Commissioning".N0169_BYPASS )
   END_RUNG
   // the same network as SCL:
   "00_Commissioning".N0169_BYPASS := "AlwaysFALSE" AND "ZAUX".N0169;
END_REGION

REGION Network 77: N0170
   // One network per node
   // TRUE if the node is not ready to be used
   // FALSE if the node is ready
   RUNG wire#powerrail
      Contact( "AlwaysFALSE" )
      Contact( "ZAUX".N0170 )
      Coil( "00_Commissioning".N0170_BYPASS )
   END_RUNG
   // the same network as SCL:
   "00_Commissioning".N0170_BYPASS := "AlwaysFALSE" AND "ZAUX".N0170;
END_REGION

REGION Network 78: N0171
   // One network per node
   // TRUE if the node is not ready to be used
   // FALSE if the node is ready
   RUNG wire#powerrail
      Contact( "AlwaysFALSE" )
      Contact( "ZAUX".N0171 )
      Coil( "00_Commissioning".N0171_BYPASS )
   END_RUNG
   // the same network as SCL:
   "00_Commissioning".N0171_BYPASS := "AlwaysFALSE" AND "ZAUX".N0171;
END_REGION

REGION Network 79: N0172
   // One network per node
   // TRUE if the node is not ready to be used
   // FALSE if the node is ready
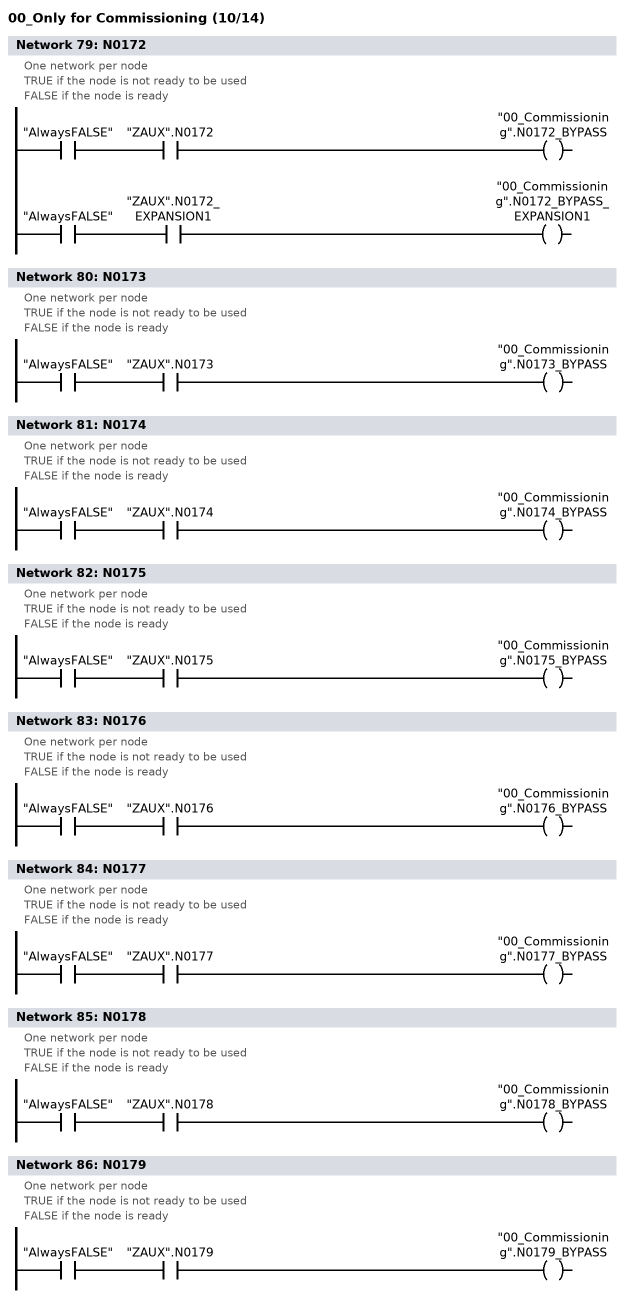
   RUNG wire#powerrail
      Contact( "AlwaysFALSE" )
      Contact( "ZAUX".N0172 )
      Coil( "00_Commissioning".N0172_BYPASS )
   END_RUNG
   RUNG wire#powerrail
      Contact( "AlwaysFALSE" )
      Contact( "ZAUX".N0172_EXPANSION1 )
      Coil( "00_Commissioning".N0172_BYPASS_EXPANSION1 )
   END_RUNG
   // the same network as SCL:
   "00_Commissioning".N0172_BYPASS := "AlwaysFALSE" AND "ZAUX".N0172;
   "00_Commissioning".N0172_BYPASS_EXPANSION1 := "AlwaysFALSE" AND "ZAUX".N0172_EXPANSION1;
END_REGION

REGION Network 80: N0173
   // One network per node
   // TRUE if the node is not ready to be used
   // FALSE if the node is ready
   RUNG wire#powerrail
      Contact( "AlwaysFALSE" )
      Contact( "ZAUX".N0173 )
      Coil( "00_Commissioning".N0173_BYPASS )
   END_RUNG
   // the same network as SCL:
   "00_Commissioning".N0173_BYPASS := "AlwaysFALSE" AND "ZAUX".N0173;
END_REGION

REGION Network 81: N0174
   // One network per node
   // TRUE if the node is not ready to be used
   // FALSE if the node is ready
   RUNG wire#powerrail
      Contact( "AlwaysFALSE" )
      Contact( "ZAUX".N0174 )
      Coil( "00_Commissioning".N0174_BYPASS )
   END_RUNG
   // the same network as SCL:
   "00_Commissioning".N0174_BYPASS := "AlwaysFALSE" AND "ZAUX".N0174;
END_REGION

REGION Network 82: N0175
   // One network per node
   // TRUE if the node is not ready to be used
   // FALSE if the node is ready
   RUNG wire#powerrail
      Contact( "AlwaysFALSE" )
      Contact( "ZAUX".N0175 )
      Coil( "00_Commissioning".N0175_BYPASS )
   END_RUNG
   // the same network as SCL:
   "00_Commissioning".N0175_BYPASS := "AlwaysFALSE" AND "ZAUX".N0175;
END_REGION

REGION Network 83: N0176
   // One network per node
   // TRUE if the node is not ready to be used
   // FALSE if the node is ready
   RUNG wire#powerrail
      Contact( "AlwaysFALSE" )
      Contact( "ZAUX".N0176 )
      Coil( "00_Commissioning".N0176_BYPASS )
   END_RUNG
   // the same network as SCL:
   "00_Commissioning".N0176_BYPASS := "AlwaysFALSE" AND "ZAUX".N0176;
END_REGION

REGION Network 84: N0177
   // One network per node
   // TRUE if the node is not ready to be used
   // FALSE if the node is ready
   RUNG wire#powerrail
      Contact( "AlwaysFALSE" )
      Contact( "ZAUX".N0177 )
      Coil( "00_Commissioning".N0177_BYPASS )
   END_RUNG
   // the same network as SCL:
   "00_Commissioning".N0177_BYPASS := "AlwaysFALSE" AND "ZAUX".N0177;
END_REGION

REGION Network 85: N0178
   // One network per node
   // TRUE if the node is not ready to be used
   // FALSE if the node is ready
   RUNG wire#powerrail
      Contact( "AlwaysFALSE" )
      Contact( "ZAUX".N0178 )
      Coil( "00_Commissioning".N0178_BYPASS )
   END_RUNG
   // the same network as SCL:
   "00_Commissioning".N0178_BYPASS := "AlwaysFALSE" AND "ZAUX".N0178;
END_REGION

REGION Network 86: N0179
   // One network per node
   // TRUE if the node is not ready to be used
   // FALSE if the node is ready
   RUNG wire#powerrail
      Contact( "AlwaysFALSE" )
      Contact( "ZAUX".N0179 )
      Coil( "00_Commissioning".N0179_BYPASS )
   END_RUNG
   // the same network as SCL:
   "00_Commissioning".N0179_BYPASS := "AlwaysFALSE" AND "ZAUX".N0179;
END_REGION

REGION Network 87: N0180
   // One network per node
   // TRUE if the node is not ready to be used
   // FALSE if the node is ready
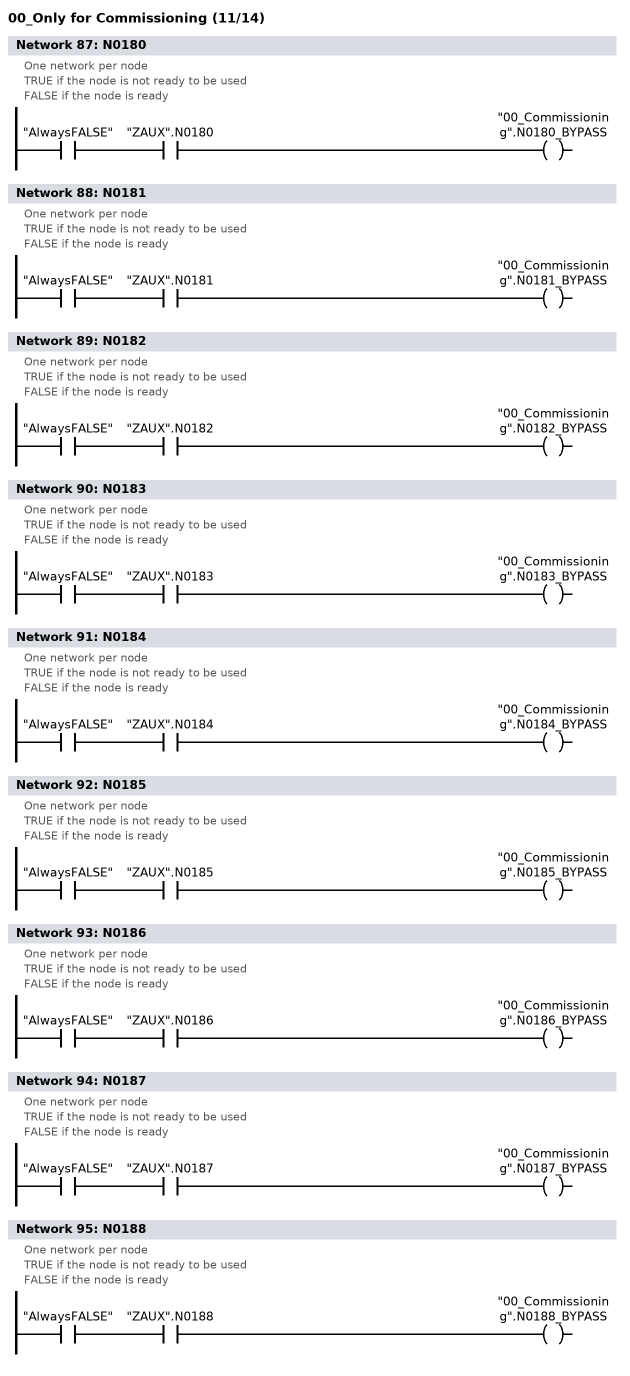
   RUNG wire#powerrail
      Contact( "AlwaysFALSE" )
      Contact( "ZAUX".N0180 )
      Coil( "00_Commissioning".N0180_BYPASS )
   END_RUNG
   // the same network as SCL:
   "00_Commissioning".N0180_BYPASS := "AlwaysFALSE" AND "ZAUX".N0180;
END_REGION

REGION Network 88: N0181
   // One network per node
   // TRUE if the node is not ready to be used
   // FALSE if the node is ready
   RUNG wire#powerrail
      Contact( "AlwaysFALSE" )
      Contact( "ZAUX".N0181 )
      Coil( "00_Commissioning".N0181_BYPASS )
   END_RUNG
   // the same network as SCL:
   "00_Commissioning".N0181_BYPASS := "AlwaysFALSE" AND "ZAUX".N0181;
END_REGION

REGION Network 89: N0182
   // One network per node
   // TRUE if the node is not ready to be used
   // FALSE if the node is ready
   RUNG wire#powerrail
      Contact( "AlwaysFALSE" )
      Contact( "ZAUX".N0182 )
      Coil( "00_Commissioning".N0182_BYPASS )
   END_RUNG
   // the same network as SCL:
   "00_Commissioning".N0182_BYPASS := "AlwaysFALSE" AND "ZAUX".N0182;
END_REGION

REGION Network 90: N0183
   // One network per node
   // TRUE if the node is not ready to be used
   // FALSE if the node is ready
   RUNG wire#powerrail
      Contact( "AlwaysFALSE" )
      Contact( "ZAUX".N0183 )
      Coil( "00_Commissioning".N0183_BYPASS )
   END_RUNG
   // the same network as SCL:
   "00_Commissioning".N0183_BYPASS := "AlwaysFALSE" AND "ZAUX".N0183;
END_REGION

REGION Network 91: N0184
   // One network per node
   // TRUE if the node is not ready to be used
   // FALSE if the node is ready
   RUNG wire#powerrail
      Contact( "AlwaysFALSE" )
      Contact( "ZAUX".N0184 )
      Coil( "00_Commissioning".N0184_BYPASS )
   END_RUNG
   // the same network as SCL:
   "00_Commissioning".N0184_BYPASS := "AlwaysFALSE" AND "ZAUX".N0184;
END_REGION

REGION Network 92: N0185
   // One network per node
   // TRUE if the node is not ready to be used
   // FALSE if the node is ready
   RUNG wire#powerrail
      Contact( "AlwaysFALSE" )
      Contact( "ZAUX".N0185 )
      Coil( "00_Commissioning".N0185_BYPASS )
   END_RUNG
   // the same network as SCL:
   "00_Commissioning".N0185_BYPASS := "AlwaysFALSE" AND "ZAUX".N0185;
END_REGION

REGION Network 93: N0186
   // One network per node
   // TRUE if the node is not ready to be used
   // FALSE if the node is ready
   RUNG wire#powerrail
      Contact( "AlwaysFALSE" )
      Contact( "ZAUX".N0186 )
      Coil( "00_Commissioning".N0186_BYPASS )
   END_RUNG
   // the same network as SCL:
   "00_Commissioning".N0186_BYPASS := "AlwaysFALSE" AND "ZAUX".N0186;
END_REGION

REGION Network 94: N0187
   // One network per node
   // TRUE if the node is not ready to be used
   // FALSE if the node is ready
   RUNG wire#powerrail
      Contact( "AlwaysFALSE" )
      Contact( "ZAUX".N0187 )
      Coil( "00_Commissioning".N0187_BYPASS )
   END_RUNG
   // the same network as SCL:
   "00_Commissioning".N0187_BYPASS := "AlwaysFALSE" AND "ZAUX".N0187;
END_REGION

REGION Network 95: N0188
   // One network per node
   // TRUE if the node is not ready to be used
   // FALSE if the node is ready
   RUNG wire#powerrail
      Contact( "AlwaysFALSE" )
      Contact( "ZAUX".N0188 )
      Coil( "00_Commissioning".N0188_BYPASS )
   END_RUNG
   // the same network as SCL:
   "00_Commissioning".N0188_BYPASS := "AlwaysFALSE" AND "ZAUX".N0188;
END_REGION

REGION Network 96: N0189
   // One network per node
   // TRUE if the node is not ready to be used
   // FALSE if the node is ready
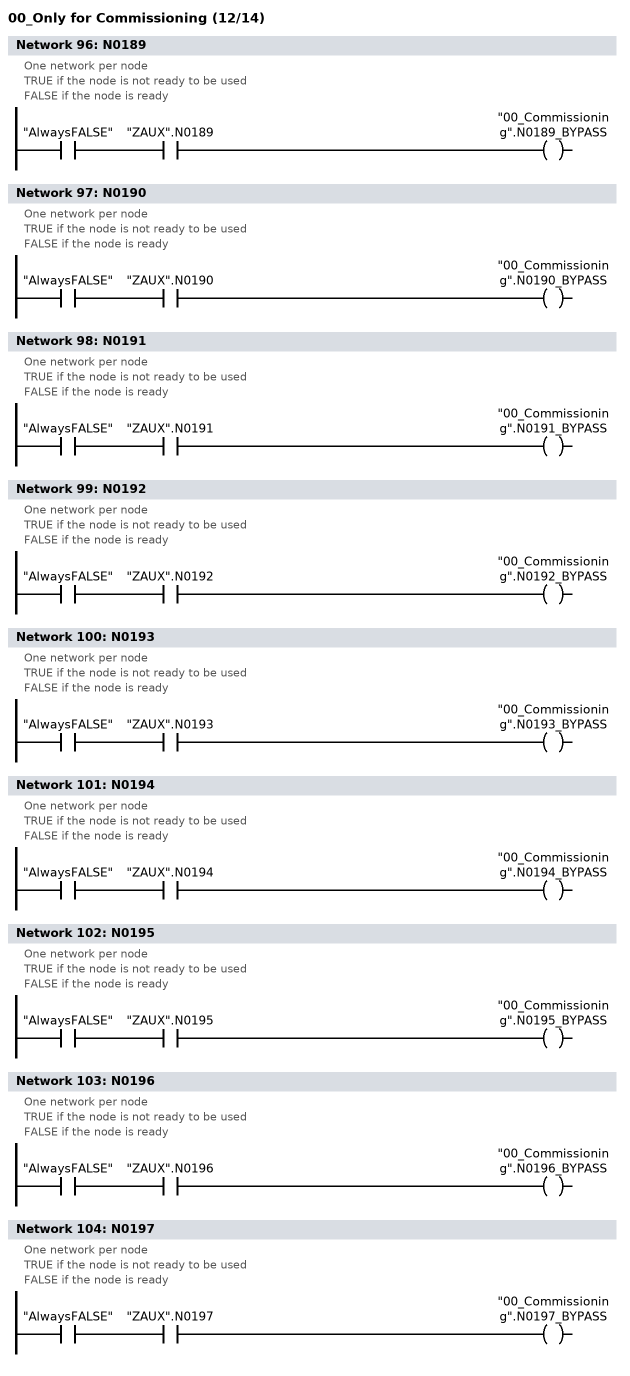
   RUNG wire#powerrail
      Contact( "AlwaysFALSE" )
      Contact( "ZAUX".N0189 )
      Coil( "00_Commissioning".N0189_BYPASS )
   END_RUNG
   // the same network as SCL:
   "00_Commissioning".N0189_BYPASS := "AlwaysFALSE" AND "ZAUX".N0189;
END_REGION

REGION Network 97: N0190
   // One network per node
   // TRUE if the node is not ready to be used
   // FALSE if the node is ready
   RUNG wire#powerrail
      Contact( "AlwaysFALSE" )
      Contact( "ZAUX".N0190 )
      Coil( "00_Commissioning".N0190_BYPASS )
   END_RUNG
   // the same network as SCL:
   "00_Commissioning".N0190_BYPASS := "AlwaysFALSE" AND "ZAUX".N0190;
END_REGION

REGION Network 98: N0191
   // One network per node
   // TRUE if the node is not ready to be used
   // FALSE if the node is ready
   RUNG wire#powerrail
      Contact( "AlwaysFALSE" )
      Contact( "ZAUX".N0191 )
      Coil( "00_Commissioning".N0191_BYPASS )
   END_RUNG
   // the same network as SCL:
   "00_Commissioning".N0191_BYPASS := "AlwaysFALSE" AND "ZAUX".N0191;
END_REGION

REGION Network 99: N0192
   // One network per node
   // TRUE if the node is not ready to be used
   // FALSE if the node is ready
   RUNG wire#powerrail
      Contact( "AlwaysFALSE" )
      Contact( "ZAUX".N0192 )
      Coil( "00_Commissioning".N0192_BYPASS )
   END_RUNG
   // the same network as SCL:
   "00_Commissioning".N0192_BYPASS := "AlwaysFALSE" AND "ZAUX".N0192;
END_REGION

REGION Network 100: N0193
   // One network per node
   // TRUE if the node is not ready to be used
   // FALSE if the node is ready
   RUNG wire#powerrail
      Contact( "AlwaysFALSE" )
      Contact( "ZAUX".N0193 )
      Coil( "00_Commissioning".N0193_BYPASS )
   END_RUNG
   // the same network as SCL:
   "00_Commissioning".N0193_BYPASS := "AlwaysFALSE" AND "ZAUX".N0193;
END_REGION

REGION Network 101: N0194
   // One network per node
   // TRUE if the node is not ready to be used
   // FALSE if the node is ready
   RUNG wire#powerrail
      Contact( "AlwaysFALSE" )
      Contact( "ZAUX".N0194 )
      Coil( "00_Commissioning".N0194_BYPASS )
   END_RUNG
   // the same network as SCL:
   "00_Commissioning".N0194_BYPASS := "AlwaysFALSE" AND "ZAUX".N0194;
END_REGION

REGION Network 102: N0195
   // One network per node
   // TRUE if the node is not ready to be used
   // FALSE if the node is ready
   RUNG wire#powerrail
      Contact( "AlwaysFALSE" )
      Contact( "ZAUX".N0195 )
      Coil( "00_Commissioning".N0195_BYPASS )
   END_RUNG
   // the same network as SCL:
   "00_Commissioning".N0195_BYPASS := "AlwaysFALSE" AND "ZAUX".N0195;
END_REGION

REGION Network 103: N0196
   // One network per node
   // TRUE if the node is not ready to be used
   // FALSE if the node is ready
   RUNG wire#powerrail
      Contact( "AlwaysFALSE" )
      Contact( "ZAUX".N0196 )
      Coil( "00_Commissioning".N0196_BYPASS )
   END_RUNG
   // the same network as SCL:
   "00_Commissioning".N0196_BYPASS := "AlwaysFALSE" AND "ZAUX".N0196;
END_REGION

REGION Network 104: N0197
   // One network per node
   // TRUE if the node is not ready to be used
   // FALSE if the node is ready
   RUNG wire#powerrail
      Contact( "AlwaysFALSE" )
      Contact( "ZAUX".N0197 )
      Coil( "00_Commissioning".N0197_BYPASS )
   END_RUNG
   // the same network as SCL:
   "00_Commissioning".N0197_BYPASS := "AlwaysFALSE" AND "ZAUX".N0197;
END_REGION

REGION Network 105: N0240
   // One network per node
   // TRUE if the node is not ready to be used
   // FALSE if the node is ready
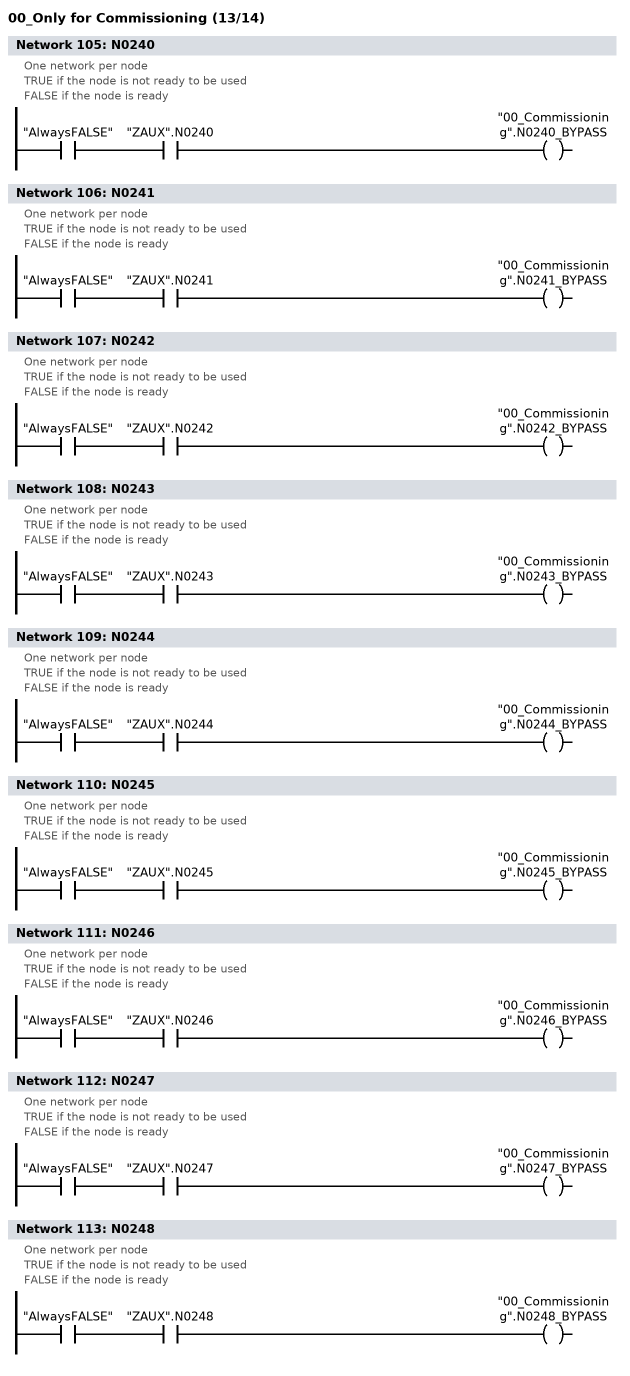
   RUNG wire#powerrail
      Contact( "AlwaysFALSE" )
      Contact( "ZAUX".N0240 )
      Coil( "00_Commissioning".N0240_BYPASS )
   END_RUNG
   // the same network as SCL:
   "00_Commissioning".N0240_BYPASS := "AlwaysFALSE" AND "ZAUX".N0240;
END_REGION

REGION Network 106: N0241
   // One network per node
   // TRUE if the node is not ready to be used
   // FALSE if the node is ready
   RUNG wire#powerrail
      Contact( "AlwaysFALSE" )
      Contact( "ZAUX".N0241 )
      Coil( "00_Commissioning".N0241_BYPASS )
   END_RUNG
   // the same network as SCL:
   "00_Commissioning".N0241_BYPASS := "AlwaysFALSE" AND "ZAUX".N0241;
END_REGION

REGION Network 107: N0242
   // One network per node
   // TRUE if the node is not ready to be used
   // FALSE if the node is ready
   RUNG wire#powerrail
      Contact( "AlwaysFALSE" )
      Contact( "ZAUX".N0242 )
      Coil( "00_Commissioning".N0242_BYPASS )
   END_RUNG
   // the same network as SCL:
   "00_Commissioning".N0242_BYPASS := "AlwaysFALSE" AND "ZAUX".N0242;
END_REGION

REGION Network 108: N0243
   // One network per node
   // TRUE if the node is not ready to be used
   // FALSE if the node is ready
   RUNG wire#powerrail
      Contact( "AlwaysFALSE" )
      Contact( "ZAUX".N0243 )
      Coil( "00_Commissioning".N0243_BYPASS )
   END_RUNG
   // the same network as SCL:
   "00_Commissioning".N0243_BYPASS := "AlwaysFALSE" AND "ZAUX".N0243;
END_REGION

REGION Network 109: N0244
   // One network per node
   // TRUE if the node is not ready to be used
   // FALSE if the node is ready
   RUNG wire#powerrail
      Contact( "AlwaysFALSE" )
      Contact( "ZAUX".N0244 )
      Coil( "00_Commissioning".N0244_BYPASS )
   END_RUNG
   // the same network as SCL:
   "00_Commissioning".N0244_BYPASS := "AlwaysFALSE" AND "ZAUX".N0244;
END_REGION

REGION Network 110: N0245
   // One network per node
   // TRUE if the node is not ready to be used
   // FALSE if the node is ready
   RUNG wire#powerrail
      Contact( "AlwaysFALSE" )
      Contact( "ZAUX".N0245 )
      Coil( "00_Commissioning".N0245_BYPASS )
   END_RUNG
   // the same network as SCL:
   "00_Commissioning".N0245_BYPASS := "AlwaysFALSE" AND "ZAUX".N0245;
END_REGION

REGION Network 111: N0246
   // One network per node
   // TRUE if the node is not ready to be used
   // FALSE if the node is ready
   RUNG wire#powerrail
      Contact( "AlwaysFALSE" )
      Contact( "ZAUX".N0246 )
      Coil( "00_Commissioning".N0246_BYPASS )
   END_RUNG
   // the same network as SCL:
   "00_Commissioning".N0246_BYPASS := "AlwaysFALSE" AND "ZAUX".N0246;
END_REGION

REGION Network 112: N0247
   // One network per node
   // TRUE if the node is not ready to be used
   // FALSE if the node is ready
   RUNG wire#powerrail
      Contact( "AlwaysFALSE" )
      Contact( "ZAUX".N0247 )
      Coil( "00_Commissioning".N0247_BYPASS )
   END_RUNG
   // the same network as SCL:
   "00_Commissioning".N0247_BYPASS := "AlwaysFALSE" AND "ZAUX".N0247;
END_REGION

REGION Network 113: N0248
   // One network per node
   // TRUE if the node is not ready to be used
   // FALSE if the node is ready
   RUNG wire#powerrail
      Contact( "AlwaysFALSE" )
      Contact( "ZAUX".N0248 )
      Coil( "00_Commissioning".N0248_BYPASS )
   END_RUNG
   // the same network as SCL:
   "00_Commissioning".N0248_BYPASS := "AlwaysFALSE" AND "ZAUX".N0248;
END_REGION

REGION Network 114: N0249
   // One network per node
   // TRUE if the node is not ready to be used
   // FALSE if the node is ready
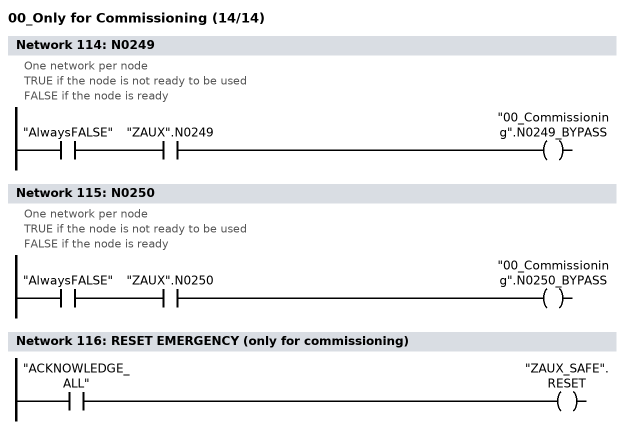
   RUNG wire#powerrail
      Contact( "AlwaysFALSE" )
      Contact( "ZAUX".N0249 )
      Coil( "00_Commissioning".N0249_BYPASS )
   END_RUNG
   // the same network as SCL:
   "00_Commissioning".N0249_BYPASS := "AlwaysFALSE" AND "ZAUX".N0249;
END_REGION

REGION Network 115: N0250
   // One network per node
   // TRUE if the node is not ready to be used
   // FALSE if the node is ready
   RUNG wire#powerrail
      Contact( "AlwaysFALSE" )
      Contact( "ZAUX".N0250 )
      Coil( "00_Commissioning".N0250_BYPASS )
   END_RUNG
   // the same network as SCL:
   "00_Commissioning".N0250_BYPASS := "AlwaysFALSE" AND "ZAUX".N0250;
END_REGION

REGION Network 116: RESET EMERGENCY (only for commissioning)
   RUNG wire#powerrail
      Contact( "ACKNOWLEDGE_ALL" )
      Coil( "ZAUX_SAFE".RESET )
   END_RUNG
   // the same network as SCL:
   "ZAUX_SAFE".RESET := "ACKNOWLEDGE_ALL";
END_REGION
END_FUNCTION
